Universal Robots PolyScope program: sendPath.urp

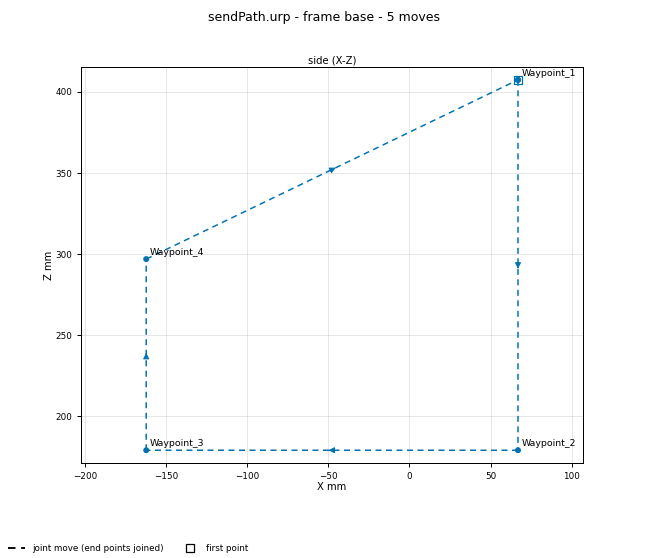
[picture p0: tool path of sendPath.urp in frame base, 5 of 5 moves have a stored position in this frame; points joined in program order, loops and branches not executed]
Program sendPath (installation=default directory=/programs/RemoteOperation createdIn=5.10.0.106268 lastSavedIn=5.10.0.106268 robotSerialNumber=20185500191)
Calibrated DH parameters: a=[0.000131, -0.165639, -0.102041, 0.000082, 0.000046, 0]; d=[0.162455, 220.258006, 1988.136334, -2208.260978, 0.099826, 0.099896]; alpha=[1.570482, -0.001777, -0.000172, 1.570393, -1.570735, 0]; deltaTheta=[0, -1.170526, -0.137148, 1.307669, -0.000001, 0]
Robot Program (runOnlyOnce=true)
  Script: write_output_integer_register(0,0)
  Wait DigitalInput pin=digital_in[0]; digitalValue=1
  MoveJ speed 15 deg/s, acceleration 30 deg/s^2 (useActiveTCP=true) feature=Base
    Waypoint Waypoint_1: TCP in base x=66.895 y=-541.759 z=407.413 mm, rx=2.1914 ry=2.251 rz=-0.0001 rad; joints [-68.793, -96.624, -69.103, -104.271, 89.915, 109.668] deg; TCP offset x=0 y=0 z=174 mm, rx=0 ry=0 rz=0 rad
    Waypoint Waypoint_2: TCP in base x=66.891 y=-541.744 z=179.168 mm, rx=2.1915 ry=2.251 rz=-0.0001 rad; joints [-68.824, -98.011, -101.373, -70.616, 89.919, 109.635] deg
    Waypoint Waypoint_3: TCP in base x=-162.208 y=-541.76 z=179.175 mm, rx=2.1914 ry=2.251 rz=-0.0001 rad; joints [-93.029, -100.628, -98.271, -71.099, 89.919, 85.424] deg
    Waypoint Waypoint_4: TCP in base x=-162.213 y=-541.753 z=296.958 mm, rx=-2.1915 ry=-2.251 rz=0 rad; joints [-93.017, -97.766, -84.084, -88.155, 89.917, 85.443] deg
    Waypoint Waypoint_1: TCP in base x=66.895 y=-541.759 z=407.413 mm, rx=2.1914 ry=2.251 rz=-0.0001 rad; joints [-68.793, -96.624, -69.103, -104.271, 89.915, 109.668] deg
  Script: write_output_integer_register(0,1)
